{attribute addProperty BoxType "AT2041-0250-0022"}
{attribute addProperty Id "A_0100_AT2040_5250_0019_AT2040_5250AT2040_3DCFC8D064080"}
{attribute addProperty CRC "3990938036"}
{attribute addProperty SizeInBites "640"}
{attribute addProperty SizeInBytes "80"}
TYPE A_0044_AT2041_0250_0022_EDE0E1B4 EXTENDS AT2041_9506A482 :
STRUCT
	{attribute addProperty Name "A_0100_AT2040_5250_0019_AT2040_5250"}
	A_0100_AT2040_5250_0019_AT2040_5250 : AT2040_3DCFC8D0;
END_STRUCT
END_TYPE

(* stored: Version 1.2.0.0, ProductVersion 3.1.4024.9
   DUT A_0044_AT2041_0250_0022_EDE0E1B4: Id {08620ec9-a3dc-4592-a1d1-8831b5744cf6} *)
